// TIA Portal V20 export
FUNCTION_BLOCK "FB_Digital_Outputs"   // FB3, LAD
{ S7_Optimized_Access := 'TRUE' }
// stored: MemoryReserve 100, SetENOAutomatically false
   VAR_INPUT
      DB_Digital_Output_0 : Bool;
      DB_Digital_Output_1 : Bool;
      DB_Digital_Output_2 : Bool;
      DB_Digital_Output_3 : Bool;
      DB_Digital_Output_4 : Bool;
      DB_Digital_Output_5 : Bool;
      DB_Digital_Output_6 : Bool;
      DB_Digital_Output_7 : Bool;
      DB_Digital_Output_8 : Bool;
      DB_Digital_Output_9 : Bool;
   END_VAR
   VAR_OUTPUT
      Q_Digital_Output_0 : Bool;
      Q_Digital_Output_1 : Bool;
      Q_Digital_Output_2 : Bool;
      Q_Digital_Output_3 : Bool;
      Q_Digital_Output_4 : Bool;
      Q_Digital_Output_5 : Bool;
      Q_Digital_Output_6 : Bool;
      Q_Digital_Output_7 : Bool;
      Q_Digital_Output_8 : Bool;
      Q_Digital_Output_9 : Bool;
   END_VAR
BEGIN

REGION Network 1
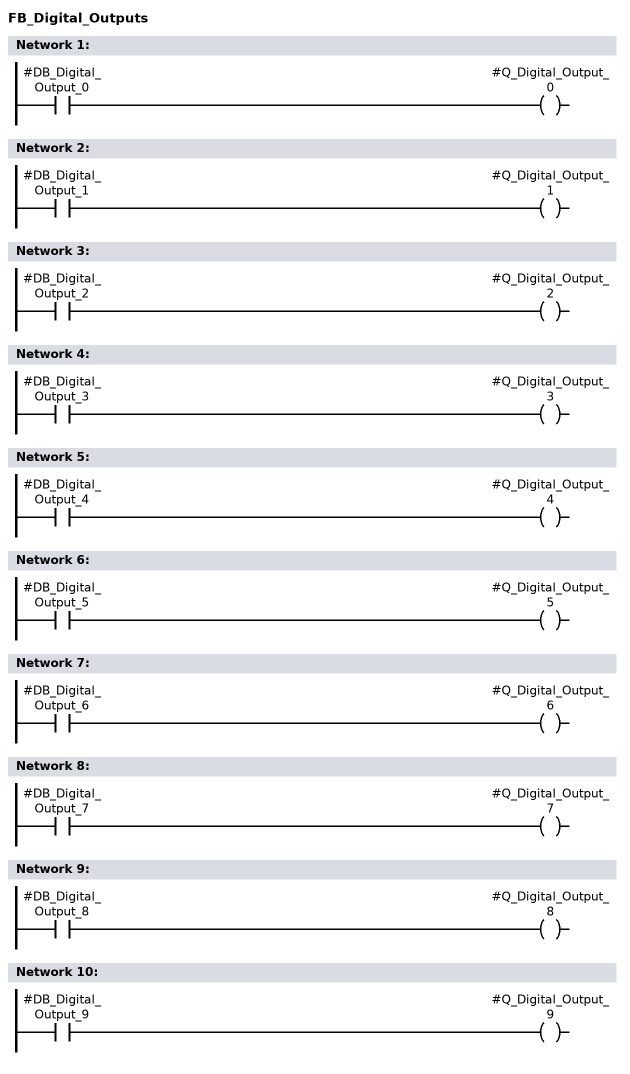
   RUNG wire#powerrail
      Contact( #DB_Digital_Output_0 )
      Coil( #Q_Digital_Output_0 )
   END_RUNG
   // the same network as SCL:
   #Q_Digital_Output_0 := #DB_Digital_Output_0;
END_REGION

REGION Network 2
   RUNG wire#powerrail
      Contact( #DB_Digital_Output_1 )
      Coil( #Q_Digital_Output_1 )
   END_RUNG
   // the same network as SCL:
   #Q_Digital_Output_1 := #DB_Digital_Output_1;
END_REGION

REGION Network 3
   RUNG wire#powerrail
      Contact( #DB_Digital_Output_2 )
      Coil( #Q_Digital_Output_2 )
   END_RUNG
   // the same network as SCL:
   #Q_Digital_Output_2 := #DB_Digital_Output_2;
END_REGION

REGION Network 4
   RUNG wire#powerrail
      Contact( #DB_Digital_Output_3 )
      Coil( #Q_Digital_Output_3 )
   END_RUNG
   // the same network as SCL:
   #Q_Digital_Output_3 := #DB_Digital_Output_3;
END_REGION

REGION Network 5
   RUNG wire#powerrail
      Contact( #DB_Digital_Output_4 )
      Coil( #Q_Digital_Output_4 )
   END_RUNG
   // the same network as SCL:
   #Q_Digital_Output_4 := #DB_Digital_Output_4;
END_REGION

REGION Network 6
   RUNG wire#powerrail
      Contact( #DB_Digital_Output_5 )
      Coil( #Q_Digital_Output_5 )
   END_RUNG
   // the same network as SCL:
   #Q_Digital_Output_5 := #DB_Digital_Output_5;
END_REGION

REGION Network 7
   RUNG wire#powerrail
      Contact( #DB_Digital_Output_6 )
      Coil( #Q_Digital_Output_6 )
   END_RUNG
   // the same network as SCL:
   #Q_Digital_Output_6 := #DB_Digital_Output_6;
END_REGION

REGION Network 8
   RUNG wire#powerrail
      Contact( #DB_Digital_Output_7 )
      Coil( #Q_Digital_Output_7 )
   END_RUNG
   // the same network as SCL:
   #Q_Digital_Output_7 := #DB_Digital_Output_7;
END_REGION

REGION Network 9
   RUNG wire#powerrail
      Contact( #DB_Digital_Output_8 )
      Coil( #Q_Digital_Output_8 )
   END_RUNG
   // the same network as SCL:
   #Q_Digital_Output_8 := #DB_Digital_Output_8;
END_REGION

REGION Network 10
   RUNG wire#powerrail
      Contact( #DB_Digital_Output_9 )
      Coil( #Q_Digital_Output_9 )
   END_RUNG
   // the same network as SCL:
   #Q_Digital_Output_9 := #DB_Digital_Output_9;
END_REGION
END_FUNCTION_BLOCK
